# EPICS autosave request: iocBoot/generic_motors_ioc/dbSave/XY_P7_.req
%
% BURT Request File
%
% $(P)XY:P7:  X-Y positioner #7
%

file assy.req ASSY=$(P)XY:P7
file mtr1.req MTR1=$(P)XY:mx7
file mtr1.req MTR1=$(P)XY:my7
file drv1.req DRV1=$(P)XY:X7
file drv1.req DRV1=$(P)XY:Y7
